FUNCTION_BLOCK E_TRAIN
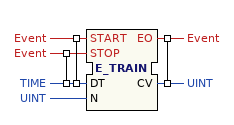
  EVENT_INPUT
    START WITH DT;
    STOP WITH DT;
  END_EVENT
  EVENT_OUTPUT
    EO WITH CV;
  END_EVENT
  VAR_INPUT
    DT : TIME;
    N : UINT;
  END_VAR
  VAR_OUTPUT
    CV : UINT;
  END_VAR
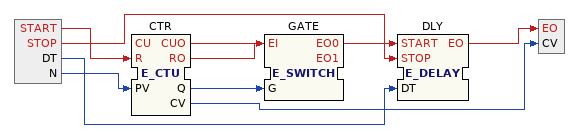
  FBS
    CTR : E_CTU;
    GATE : E_SWITCH;
    DLY : E_DELAY;
  END_FBS
  EVENT_CONNECTIONS
    CTR.CUO TO GATE.EI;
    CTR.RO TO GATE.EI;
    START TO CTR.R;
    GATE.EO0 TO DLY.START;
    STOP TO DLY.STOP;
    DLY.EO TO EO;
  END_CONNECTIONS
  DATA_CONNECTIONS
    N TO CTR.PV;
    CTR.CV TO CV;
    DT TO DLY.DT;
    CTR.Q TO GATE.G;
  END_CONNECTIONS
END_FUNCTION_BLOCK
